// TIA Portal V20 export
VAR_GLOBAL   // PLC tag table "IO"
   "I_IN1_EXT+SGV" AT %I0.0 : Bool;   // communication spare (not used)
   "I_IN2_EXT+SGV" AT %I0.1 : Bool;   // communication spare (not used)
   "I_IN3_EXT+SGV" AT %I0.2 : Bool;   // communication spare (not used)
   "I_0E1+SGV" AT %I0.3 : Bool;   // air conditioner 1 scannerhousing visual measurement (1=ok)
   "I_0E2+SGX" AT %I0.4 : Bool;   // air conditioner scannerhousing x-ray measurement (1=ok)
   "I_0F1.1+SGV" AT %I0.5 : Bool;   // monitoring circuit breaker supply 24V ( -0F1.1)
   "I_0SH1+SSTR" AT %I0.6 : Bool;   // cooling fan / air conditioner off (cleaning filter)
   "I_14SB0+HMI" AT %I0.7 : Bool;   // emergency stop Goldeneye HMI
   "I_14SB1+HMI" AT %I1.0 : Bool;   // scanner release Goldeneye HMI
   "I_8S1.T_in" AT %I1.1 : Bool;   // adjustment top limit switch innermost position
   "I_8S2.T_out" AT %I1.2 : Bool;   // adjustment top limit switch outermost position
   "I_8S1.L_in" AT %I1.3 : Bool;   // adjustment left limit switch innermost position
   "I_8S2.L_out" AT %I1.4 : Bool;   // adjustment left limit switch outermost position
   "I_8S1.R_in" AT %I1.5 : Bool;   // adjustment right limit switch innermost position
   "I_8S2.R_out" AT %I1.6 : Bool;   // adjustment right limit switch outermost position
   "I_8S1.B_left" AT %I2.0 : Bool;   // adjustment scannerhousing limit switch left position
   "I_8S2.B_right" AT %I2.1 : Bool;   // adjustment scannerhousing limit switch right position
   "I_1BTR2+SGX" AT %I2.2 : Bool;   // light barrier in scannerhousing x-ray measurement
   "O_14VK1+SGV" AT %Q0.0 : Bool;   // safety loops scanner internal ok
   "O_14VK2+SGV" AT %Q0.1 : Bool;   // setting mode active
   "O_0VK1+SGV" AT %Q0.2 : Bool;   // scanner ready
   "O_0VK2+SGV" AT %Q0.3 : Bool;   // scanner error
   "O_0VK3+SGV" AT %Q0.4 : Bool;   // communication spare (not used)
   "O_0VK4+SGV" AT %Q0.5 : Bool;   // communication spare (not used)
   "O_0F1.1+SGV" AT %Q0.6 : Bool;   // acknowledge circuit breaker supply 24V
   "O_0KA0.1+SGV" AT %Q0.7 : Bool;   // air conditioner scannerhousing visual measurement off
   "O_0KA1+SGV" AT %Q1.1 : Bool;   // scanner status display
   "O_8M1.T_c" AT %Q1.2 : Bool;   // adjustment top close
   "O_8M1.T_o" AT %Q1.3 : Bool;   // adjustment top open
   "O_8M1.L_c" AT %Q1.4 : Bool;   // adjustment left close
   "O_8M1.L_o" AT %Q1.5 : Bool;   // adjustment left open
   "O_8M1.R_c" AT %Q1.6 : Bool;   // adjustment right close
   "O_8M1.R_o" AT %Q1.7 : Bool;   // adjustment right open
   "O_8M1.B_l" AT %Q2.1 : Bool;   // adjustment scannerhousing left
   "O_8M1.B_r" AT %Q2.2 : Bool;   // adjustment scannerhousing right
   "SI_NA_EXT+SGV" AT %I800.0 : Bool;   // emergency stop + area stop external
   "SI_14SB0/1+HMI" AT %I800.1 : Bool;   // emergency stop / scanner release Goldeneye HMI
   "SI_14SB1+SSTL" AT %I800.2 : Bool;   // setting mode scanner active
   "SI_14SB2+SSTL" AT %I800.3 : Bool;   // jog adjustment camera
   "SI_8U1+SGV" AT %I824.0 : Bool;   // adjustment linear drive monitoring
   "SI_14KA1+SGV" AT %I824.1 : Bool;   // area laser monitoring
   "SI_14KA2+SGV" AT %I824.2 : Bool;   // area adjustment monitoring
   "SI_14SS1.TL+SGV" AT %I808.0 : Bool;   // safety contact cover top left SGV
   "SI_14SS1.BL+SGV" AT %I808.1 : Bool;   // safety contact cover bottom left SGV
   "SI_14SS1.TR+SGV" AT %I808.2 : Bool;   // safety contact cover top right SGV
   "SI_14SS1.BR+SGV" AT %I808.3 : Bool;   // safety contact cover bottom right SGV
   "SI_14SS1.TL+SGX" AT %I816.0 : Bool;   // safety contact cover top left SGX
   "SI_14SS1.BL+SGX" AT %I816.1 : Bool;   // safety contact cover bottom left SGX
   "SI_14SS1.TR+SGX" AT %I816.2 : Bool;   // safety contact cover top right SGX
   "SI_14SS1.BR+SGX" AT %I816.3 : Bool;   // safety contact cover bottom right SGX
   "SO_14HV1+SSTL/R" AT %Q900.1 : Bool;   // setting mode scanner active
   "SO_14KA1+SGV" AT %Q900.2 : Bool;   // area laser on
   "SO_14KA2+SGV" AT %Q900.3 : Bool;   // area adjustment on
   "SO_ST.3HF+SGV" AT %Q908.0 : Bool;   // safety lamp laser on
   "SO_ST.5HF+SGV" AT %Q908.1 : Bool;   // safety lamp X-Ray on
   "SO_5AX1+SGX" AT %Q908.2 : Bool;   // area x-ray on
   "O_8KA1+SGV" AT %Q2.0 : Bool;   // adjustment linear drive reset (not used)
   "I_1BTR2+SGV" AT %I1.7 : Bool;   // light barrier in scannerhousing visual measurement
   "O_2YV1/2.B+SGV" AT %Q2.3 : Bool;   // blow-off valve SGV bottom
   "O_2YV1.L+SGV" AT %Q2.4 : Bool;   // blow-off valve SGV left
   "O_2YV1.R+SGV" AT %Q2.5 : Bool;   // blow-off valve SGV right
   "O_5YV1+SGX" AT %Q2.6 : Bool;   // blow-off valve SGX X-Ray
   "O_0KA0.2+SGV" AT %Q1.0 : Bool;   // air conditioner scannerhousing x-ray measurement off
   "SI_5AX1+SGX" AT %I824.3 : Bool;   // area x-ray monitoring
   O_spare27 AT %Q2.7 : Bool;   // output normal spare
   "I_0E1.1+SGV" AT %I2.3 : Bool;   // air conditioner 2 scannerhousing visual measurement (1=ok)
   I_spare24 AT %I2.4 : Bool;
   I_spare25 AT %I2.5 : Bool;
   I_spare26 AT %I2.6 : Bool;
   I_spare27 AT %I2.7 : Bool;
   SO_spare9083 AT %Q908.3 : Bool;
   SO_safetynew AT %Q900.0 : Bool;
   I_test AT %I5.0 : Bool;
END_VAR
